TYPE (* A Structure with 1 Bit *)
  (* Version 1.0, 2024-02-21, franz *)
  PACKAGE bits;
  st1b : STRUCT
    b0 : BOOL; (* BIT 00 *)
  END_STRUCT;
END_TYPE
